{attribute 'pack_mode' := '2'}
TYPE ST_STATION_STATE :
STRUCT
  eState          : E_STATION_STATE;
  {attribute 'displaymode':='bin'}
  nMask           : BYTE;
  nMoverId        : USINT;
  rMoverModPos    : lreal; // modulo position of detected mover
  nQueue          : USINT; // queue count for station
END_STRUCT
END_TYPE

(* stored: Version 1.1.0.1, ProductVersion 3.1.4024.12
   DUT ST_STATION_STATE: Id {1ae51e1e-c69e-4416-bbd9-899aa6a35a6b} *)
